{attribute addProperty BoxType "EL5101-0011-0016"}
{attribute addProperty Id "Counter_valueAT %I*ARRAY [0..0] OF UDINT324"}
{attribute addProperty CRC "1929918584"}
{attribute addProperty SizeInBites "32"}
{attribute addProperty SizeInBytes "4"}
TYPE ENC_TxPdo_1_Samples_Counter_value_73083878 :
STRUCT
	{attribute addProperty Name "Counter_value"}
	Counter_value AT %I* : ARRAY [0..0] OF UDINT;
END_STRUCT
END_TYPE

(* stored: Version 1.2.0.0, ProductVersion 3.1.4024.9
   DUT ENC_TxPdo_1_Samples_Counter_value_73083878: Id {d4fe07fa-53b0-47a6-9b97-31ac85103e59} *)
